INTERFACE I_State EXTENDS __SYSTEM.IQueryInterface

METHOD OnEntry
VAR_INPUT
END_VAR
END_METHOD

METHOD OnExit
VAR_INPUT
END_VAR
END_METHOD

END_INTERFACE

(* stored: Version 1.1.0.1, ProductVersion 3.1.4024.12
   Itf I_State: Id {d0774aa8-d167-42f9-abda-f16771fab9bf}
   Method OnEntry: Id {0c43d4ef-c2ed-49c7-b57a-e9530adbb5a1}
   Method OnExit: Id {178599ec-0942-4cf4-a9df-f753f7c04af7} *)
